# EPICS autosave request: iocBoot/iocsrsDS345/auto_settings.req
file srsDS345_settings.req P=$(P)
